TYPE ST_ActuatorOutputs :
STRUCT
	Advance  AT%Q* : BOOL;
	Retract  AT%Q* : BOOL;
END_STRUCT
END_TYPE

(* stored: Version 1.1.0.1, ProductVersion 3.1.4024.12
   DUT ST_ActuatorOutputs: Id {d02a17fe-dcc7-4240-b862-706a352f9a1a} *)
